FUNCTION_BLOCK E_D_FF_5 (* Data latch (d) flip flop for 5 BOOLs, EO only on change of at least one (generic FB) *)
  (* Standard: 61499-1 Annex A; Description: Copyright (c) 2017, 2026 fortiss GmbH, HR Agrartechnik GmbH This program and the accompanying materials are made available under the terms of the Eclipse Public License 2.0 which is available at https://www.eclipse.org/legal/epl-2.0/ SPDX-License-Identifier: EPL-2.0 *)
  (* Version 1.0, 2026-08-26, Franz Höpfinger, HR Agrartechnik GmbH, E_D_FF extended to 5 BOOLs - EO fires only if at least one Di differs from the latched Qi. Service Interface FB, native implementation GEN_E_D_FF (FORTE) required. *)
  PACKAGE iec61499::events;
  {SET_ATTRIBUTE(eclipse4diac::core::GenericClassName, 'GEN_E_D_FF')}
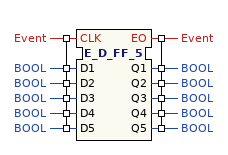
  EVENT_INPUT
    CLK WITH D1, D2, D3, D4, D5; (* Clock *)
  END_EVENT
  EVENT_OUTPUT
    EO WITH Q1, Q2, Q3, Q4, Q5; (* Triggered if clock results in a change of at least one Q *)
  END_EVENT
  VAR_INPUT
    D1 : BOOL; (* Value 1 to latch *)
    D2 : BOOL; (* Value 2 to latch *)
    D3 : BOOL; (* Value 3 to latch *)
    D4 : BOOL; (* Value 4 to latch *)
    D5 : BOOL; (* Value 5 to latch *)
  END_VAR
  VAR_OUTPUT
    Q1 : BOOL; (* Latched value 1 *)
    Q2 : BOOL; (* Latched value 2 *)
    Q3 : BOOL; (* Latched value 3 *)
    Q4 : BOOL; (* Latched value 4 *)
    Q5 : BOOL; (* Latched value 5 *)
  END_VAR
END_FUNCTION_BLOCK
